TYPE ST_AteqBitmap :
STRUCT
	stCommands 				: ST_AteqCommands;
	stEcho					: ST_AteqEcho;
	stErrorCode				: ST_AteqErrorCode;
	stRealtimeTestResults	: ST_AteqRealtimeTestResults;
END_STRUCT
END_TYPE

(* stored: Version 1.1.0.1, ProductVersion 3.1.4024.15
   DUT ST_AteqBitmap: Id {51deaec3-f483-42cf-82c8-ee242ea32ecc} *)
